(* IEC 61131-3 sources: CodesysTest/export/ObjectHandling/FB_CollectionHandleMachineComponents.pou, 9 files *)

(* ---- FB_CollectionHandleMachineComponents.pou.st ---- *)
(*#-#-#-#-#-#-#-#-#-#---Declaration---#-#-#-#-#-#-#-#-#-#-#-#-#*)

FUNCTION_BLOCK FB_CollectionHandleMachineComponents
VAR_INPUT
END_VAR
VAR
	Collection: ARRAY[0..GlobalObjects.MAX_COMPONENTS] OF IComponent; // object array
	ObjNames   : ARRAY[0..GlobalObjects.MAX_COMPONENTS] OF STRING;
	ActiveState : ARRAY[0..GlobalObjects.MAX_COMPONENTS] OF STRING;
	Ready : ARRAY[0..GlobalObjects.MAX_COMPONENTS] OF BOOL;
	InUse : ARRAY[0..GlobalObjects.MAX_COMPONENTS] OF BOOL;
	_ArrayOver   : BOOL;
	_BadObj      : INT;
	_DupeObj   : INT;
	_OverObj   : INT;
	_TotalObj   : UINT;

END_VAR(*#-#-#-#-#-#-#-#-#-#---Implementation---#-#-#-#-#-#-#-#-#-#-#-#-#*)

//	Function Block: FB_CollectionHandlerExecutable
//	Description: This collection handler stores executable FB's to an array
//				 and has a method to execute them all on demand
//	Created by: Ben Hess
//	Created Date: Friday, September 7, 2018

(* ---- AddObject.m.st ---- *)
(*#-#-#-#-#-#-#-#-#-#---Declaration---#-#-#-#-#-#-#-#-#-#-#-#-#*)

METHOD AddObject
VAR_INPUT
	Obj : IComponent;
END_VAR
VAR
	I : UINT;
	J : UINT;
END_VAR(*#-#-#-#-#-#-#-#-#-#---Implementation---#-#-#-#-#-#-#-#-#-#-#-#-#*)

// Add the active fault to the array
FOR J:= 0 TO _TotalObj DO
	IF Collection[J] = Obj THEN
		// object pointer matches - it's already in here
		RETURN;
	END_IF
END_FOR

IF _TotalObj < GlobalObjects.MAX_COMPONENTS THEN
	Collection[_TotalObj]:= Obj;
	ObjNames[_TotalObj]:= Obj.InstanceName;
	_TotalObj:= _TotalObj + 1;
ELSE
	_ArrayOver:= TRUE;
	_OverObj:= _OverObj + 1;
END_IF

(* ---- CheckIfAllHomed.m.st ---- *)
(*#-#-#-#-#-#-#-#-#-#---Declaration---#-#-#-#-#-#-#-#-#-#-#-#-#*)

METHOD CheckIfAllHomed : BOOL
VAR_INPUT
END_VAR
VAR
	J : UINT;
	homed : BOOL;
END_VAR(*#-#-#-#-#-#-#-#-#-#---Implementation---#-#-#-#-#-#-#-#-#-#-#-#-#*)

// Go through list of homable components and return true if all are homed OR if component isn't active
FOR J:= 0 TO _TotalObj - 1 DO
	homed := CheckIfHomed(Collection[J]);
END_FOR
CheckIfAllHomed := homed;

(* ---- CheckIfAllReady.m.st ---- *)
(*#-#-#-#-#-#-#-#-#-#---Declaration---#-#-#-#-#-#-#-#-#-#-#-#-#*)

METHOD CheckIfAllReady : BOOL
VAR_INPUT
END_VAR
VAR
	J : UINT;
	notReady : BOOL;
END_VAR(*#-#-#-#-#-#-#-#-#-#---Implementation---#-#-#-#-#-#-#-#-#-#-#-#-#*)

// Go through list of homable components and return true if all are homed OR if component isn't active
FOR J:= 0 TO _TotalObj - 1 DO
	IF NOT CheckIfReady(Collection[J]) THEN
		notReady := TRUE;
	END_IF
END_FOR
CheckIfAllReady := NOT notReady;

(* ---- ForceHomeAll.m.st ---- *)
(*#-#-#-#-#-#-#-#-#-#---Declaration---#-#-#-#-#-#-#-#-#-#-#-#-#*)

METHOD ForceHomeAll
VAR_INPUT
END_VAR
VAR
	Cast : IHomable;
	J : UINT;
END_VAR(*#-#-#-#-#-#-#-#-#-#---Implementation---#-#-#-#-#-#-#-#-#-#-#-#-#*)

// For each homable objest in the array, run its "HomeNow()" method
FOR J:= 0 TO _TotalObj - 1 DO
	IF (__QUERYINTERFACE(Collection[J], Cast)) THEN
		Cast.HomeNow();
	END_IF
END_FOR

(* ---- HomeAll.m.st ---- *)
(*#-#-#-#-#-#-#-#-#-#---Declaration---#-#-#-#-#-#-#-#-#-#-#-#-#*)

METHOD HomeAll
VAR_INPUT
END_VAR
VAR
	Cast : IHomable;
	J : UINT;
END_VAR(*#-#-#-#-#-#-#-#-#-#---Implementation---#-#-#-#-#-#-#-#-#-#-#-#-#*)

// For each homable objest in the array, run its "HomeNow()" method if object is not homed
FOR J:= 0 TO _TotalObj - 1 DO
	IF (__QUERYINTERFACE(Collection[J], Cast)) THEN
		IF NOT Cast.IsHomed THEN
			Cast.HomeNow();
		END_IF
	END_IF
END_FOR

(* ---- MakeReadyAll.m.st ---- *)
(*#-#-#-#-#-#-#-#-#-#---Declaration---#-#-#-#-#-#-#-#-#-#-#-#-#*)

METHOD MakeReadyAll : BOOL
VAR
	J : UINT;
END_VAR
(*#-#-#-#-#-#-#-#-#-#---Implementation---#-#-#-#-#-#-#-#-#-#-#-#-#*)

// Reset all components
FOR J:= 0 TO _TotalObj - 1 DO
	IF NOT Collection[J].Ready AND Collection[j].OptionActive THEN
		Collection[J].MakeReady();
	END_IF
END_FOR

(* ---- ResetAll.m.st ---- *)
(*#-#-#-#-#-#-#-#-#-#---Declaration---#-#-#-#-#-#-#-#-#-#-#-#-#*)

METHOD ResetAll
VAR_INPUT
END_VAR
VAR
	J : UINT;
END_VAR(*#-#-#-#-#-#-#-#-#-#---Implementation---#-#-#-#-#-#-#-#-#-#-#-#-#*)

// Reset all components
FOR J:= 0 TO _TotalObj - 1 DO
	Collection[J].Reset();
END_FOR

(* ---- UpdateInfo.m.st ---- *)
(*#-#-#-#-#-#-#-#-#-#---Declaration---#-#-#-#-#-#-#-#-#-#-#-#-#*)

METHOD UpdateInfo : BOOL
VAR_INPUT
END_VAR
VAR
	J : UINT;
END_VAR(*#-#-#-#-#-#-#-#-#-#---Implementation---#-#-#-#-#-#-#-#-#-#-#-#-#*)

FOR J:= 0 TO _TotalObj - 1 DO
		ActiveState[J]:= Collection[J].StateString;
		Ready[J] :=  Collection[J].Ready;
		InUse[J] := Collection[J].OptionActive AND Collection[J].OptionEnabled;
END_FOR
